{attribute addProperty BoxType "EL5151-0021-0018"}
{attribute addProperty Id "Latch_value_rising_edgeAT %I*UDINT32423Latch_value_falling_edgeAT %I*UDINT32424"}
{attribute addProperty CRC "2137462420"}
{attribute addProperty SizeInBites "64"}
{attribute addProperty SizeInBytes "8"}
TYPE ENC_Filtered_latch_7F671694 :
STRUCT
	{attribute addProperty Name "Latch_value_rising_edge"}
	Latch_value_rising_edge AT %I* : UDINT;
	{attribute addProperty Name "Latch_value_falling_edge"}
	Latch_value_falling_edge AT %I* : UDINT;
END_STRUCT
END_TYPE

(* stored: Version 1.2.0.0, ProductVersion 3.1.4024.9
   DUT ENC_Filtered_latch_7F671694: Id {5ec85bc1-f017-480a-a5fb-6b0acec0d484} *)
